INTERFACE I_Conveyer

METHOD Start : BOOL
VAR_INPUT
END_VAR
END_METHOD

METHOD Stop : BOOL
VAR_INPUT
END_VAR
END_METHOD

END_INTERFACE

(* stored: Version 1.1.0.1, ProductVersion 3.1.4024.16
   Itf I_Conveyer: Id {8a75df41-d8f4-4212-b044-9428a92c4db6}
   Method Start: Id {10507920-303f-41ac-8a81-e5c5d73c22be}
   Method Stop: Id {96426f84-b916-422c-900c-c875f1357b2e} *)
